Universal Robots PolyScope program: Ruch8MS.urp

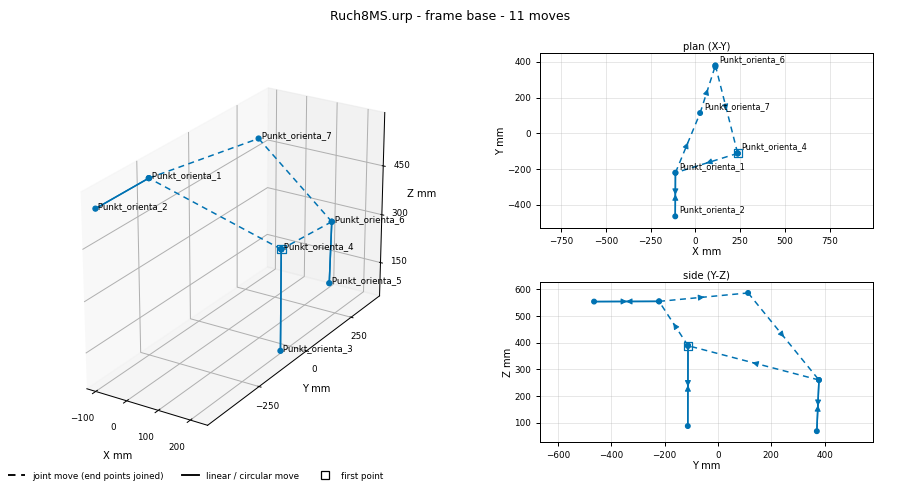
[picture p0: tool path of Ruch8MS.urp in frame base, 11 of 11 moves have a stored position in this frame; points joined in program order, loops and branches not executed]
Program Ruch8MS (installation=default directory=/programs/usbdisk createdIn=3.15.8.106339 lastSavedIn=3.15.8.106339 robotSerialNumber=2020330428)
Calibrated DH parameters: a=[0.000029, -0.241913, -0.128453, -0.000049, -0.000012, 0]; d=[0.151842, -4.082088, 33.504745, -29.309875, 0.08529, 0.082285]; alpha=[1.571059, -0.006644, 0.005794, 1.571984, -1.571997, 0]; deltaTheta=[-0.000032, 0.111537, 0.813391, -0.924919, 0.000036, 0.000016]
Robot Program (runOnlyOnce=false)
  MoveL speed 400 mm/s, acceleration 800 mm/s^2 (useActiveTCP=true) feature=Base
    Waypoint Punkt_orienta_4: TCP in base x=236.199 y=-111.927 z=388.816 mm, rx=2.2233 ry=-2.2188 rz=-0.0017 rad; joints [0.004, -89.999, -45, -135, 90, 0.002] deg; flange x=236.288 y=-111.954 z=463.816 mm, rx=2.2233 ry=-2.2188 rz=-0.0017 rad
    Waypoint Punkt_orienta_3: TCP in base x=236.723 y=-112.694 z=87.696 mm, rx=2.2254 ry=-2.2101 rz=0.0056 rad; joints [0, -90, -135, -45, 90, 0] deg; flange x=236.81 y=-112.23 z=162.695 mm, rx=2.2254 ry=-2.2101 rz=0.0056 rad
    Waypoint Punkt_orienta_4: TCP in base x=236.199 y=-111.927 z=388.816 mm, rx=2.2233 ry=-2.2188 rz=-0.0017 rad; joints [0.004, -89.999, -45, -135, 90, 0.002] deg; flange x=236.288 y=-111.954 z=463.816 mm, rx=2.2233 ry=-2.2188 rz=-0.0017 rad
  MoveJ speed 120 deg/s, acceleration 240 deg/s^2 (useActiveTCP=true)
    Waypoint Punkt_orienta_1: TCP in base x=-111.436 y=-220.479 z=554.97 mm, rx=0.0057 ry=-2.2198 rz=2.2172 rad; joints [-90, -60, -90, -30, 90, 0.002] deg; flange x=-111.406 y=-145.479 z=555.058 mm, rx=0.0057 ry=-2.2198 rz=2.2172 rad
  MoveL speed 500 mm/s, acceleration 1200 mm/s^2 (useActiveTCP=true) feature=Base
    Waypoint Punkt_orienta_2: TCP in base x=-112.454 y=-463.994 z=554.199 mm, rx=0.0008 ry=2.2221 rz=-2.2194 rad; joints [-89.999, -120, -30, -30, 90, 0.002] deg; flange x=-112.48 y=-388.995 z=554.289 mm, rx=0.0008 ry=2.2221 rz=-2.2194 rad
    Waypoint Punkt_orienta_1: TCP in base x=-111.436 y=-220.479 z=554.97 mm, rx=0.0057 ry=-2.2198 rz=2.2172 rad; joints [-90, -60, -90, -30, 90, 0.002] deg; flange x=-111.406 y=-145.479 z=555.058 mm, rx=0.0057 ry=-2.2198 rz=2.2172 rad
  MoveJ speed 200 deg/s, acceleration 400 deg/s^2 (useActiveTCP=true)
    Waypoint Punkt_orienta_7: motionParameters(blendRadius=0.236); TCP in base x=26.452 y=113.307 z=586.568 mm, rx=-1.2086 ry=-1.2149 rz=1.2179 rad; joints [-180, -90, 60, -150, 90.001, 0.004] deg; flange x=101.449 y=113.975 z=586.657 mm, rx=-1.2086 ry=-1.2149 rz=1.2179 rad
    Waypoint Punkt_orienta_6: motionParameters(blendRadius=0.1921); TCP in base x=111.869 y=378.761 z=260.382 mm, rx=3.1404 ry=0.0038 rz=0.0012 rad; joints [-270, -110, -60, -100, 89.999, 0] deg; flange x=111.809 y=378.85 z=335.382 mm, rx=3.1404 ry=0.0038 rz=0.0012 rad
  MoveL speed 500 mm/s, acceleration 1200 mm/s^2 (useActiveTCP=true) feature=Base
    Waypoint Punkt_orienta_5: TCP in base x=111.746 y=370.902 z=68.403 mm, rx=3.1404 ry=0.0094 rz=0.0042 rad; joints [-269.998, -120, -100, -50, 89.999, -0.001] deg; flange x=111.543 y=370.989 z=143.403 mm, rx=3.1404 ry=0.0094 rz=0.0042 rad
    Waypoint Punkt_orienta_8: TCP in base x=111.869 y=378.761 z=260.382 mm, rx=3.1404 ry=0.0038 rz=0.0012 rad; joints [-270, -110, -60, -100, 89.999, 0] deg; flange x=111.809 y=378.85 z=335.382 mm, rx=3.1404 ry=0.0038 rz=0.0012 rad
  MoveJ speed 240 deg/s, acceleration 480 deg/s^2 (useActiveTCP=true)
    Waypoint Punkt_orienta_4: motionParameters(blendRadius=0.05); TCP in base x=236.199 y=-111.927 z=388.816 mm, rx=2.2233 ry=-2.2188 rz=-0.0017 rad; joints [0.004, -89.999, -45, -135, 90, 0.002] deg; flange x=236.288 y=-111.954 z=463.816 mm, rx=2.2233 ry=-2.2188 rz=-0.0017 rad
